FUNCTION_BLOCK FileRemover IMPLEMENTS Cyclic
VAR
	remover : FB_FileDelete;
	
	filenameForAlarm : T_MaxString;
	removeErrorTrigger : R_TRIG;
	notFoundError : MessageEventLogger(TC_EVENTS.FileEventClass.InvalidPath);
	removeError : MessageEventLogger(TC_EVENTS.FileEventClass.RemoveFileError);
	
	removing : BOOL;
	_Done : BOOL;
END_VAR
VAR CONSTANT
	NotFoundErrorNumber : UDINT := 16#70C;
END_VAR

{attribute 'monitoring' := 'call'}
PROPERTY Busy : BOOL
GET
Busy := remover.bBusy;
END_GET
END_PROPERTY

METHOD Cyclic
remover(bExecute := FALSE);

IF (NOT remover.bBusy) THEN
	IF (NOT remover.bError AND removing) THEN
		_Done := TRUE;
	END_IF
	removing := FALSE;
END_IF

removeErrorTrigger(CLK := remover.bError);
IF (removeErrorTrigger.Q) THEN
	
	filenameForAlarm := remover.sPathName;
	IF (EventParameters.EscapeBackslash) THEN
		filenameForAlarm := ReplaceAll(filenameForAlarm, '\', '\\'); // Escape backslash to use with web-based HMIs
	END_IF
	
	IF (remover.nErrId = NotFoundErrorNumber) THEN
		notFoundError.Arguments.Clear().AddStringByValue(filenameForAlarm);
		notFoundError.Send();
	ELSE
		removeError.Arguments.Clear().AddStringByValue(filenameForAlarm);
		removeError.Send();
	END_IF
END_IF
END_METHOD

{attribute 'monitoring' := 'call'}
PROPERTY Done : BOOL
GET
Done := _Done;
END_GET
END_PROPERTY

{attribute 'monitoring' := 'call'}
PROPERTY Error : BOOL
GET
Error := remover.bError;
END_GET
END_PROPERTY

METHOD Remove
VAR_INPUT
	filePath : T_MaxString;
END_VAR
removing := TRUE;
_Done := FALSE;

remover(
	sPathName := filePath,
	bExecute := TRUE
);
END_METHOD

END_FUNCTION_BLOCK

(* stored: Version 1.1.0.1
   POU FileRemover: Id {f7631349-6fbc-06d3-2ed1-b29f37a58820}, SpecialFunc None
   Property Busy: Id {6bd9c1ba-3f65-0d10-0cde-1b0febffc27a}
   Get Get: Id {7330f990-a5d5-04b3-07af-6d657e583eb7}
   Method Cyclic: Id {e68b946e-3bea-094e-29ea-8dfdd035f074}
   Property Done: Id {8d1148ae-8a6e-029b-0ac4-e72e888d52f0}
   Get Get: Id {901f71c5-f4ad-031d-3b10-edc5b10ddbfc}
   Property Error: Id {37d95ad4-6e51-025d-1e9c-0f61cddc459e}
   Get Get: Id {c687127d-3d11-0455-00b6-d05aa4aff756}
   Method Remove: Id {b55707fa-85a0-0194-3bd7-ee768eaf1a8e} *)
